(* PLC project PLC411_AI, home PLC411_AI 1 *)
(* stored: creationDateTime 2023-04-11T09:59:45, productRelease 0, modificationDateTime 2023-04-11T09:59:45, version 1 *)

(* Установка режима работы аналогового входа *)
FUNCTION_BLOCK AIMode
  VAR_INPUT
    AIn : BYTE := 0;  (* номер входа *)
    M : BYTE := 0;  (* режим работы *)
  END_VAR
  VAR_OUTPUT
    Om : BYTE := 0;  (* режим работы (установленный) *)
    Os : BYTE := 0;  (* код состояния входа *)
    Ok : BYTE := 0;  (* код результата исполнения блока *)
  END_VAR

            {extern void App_AIMode(AIMODE*);App_AIMode(data__);}

          
END_FUNCTION_BLOCK

(* Получение значения аналогового входа *)
FUNCTION_BLOCK AINorm
  VAR_INPUT
    AIn : BYTE := 0;  (* номер входа *)
  END_VAR
  VAR_OUTPUT
    Ov : REAL := 0.0;  (* значение *)
    Os : BYTE := 0;  (* код состояния *)
    Ok : BYTE := 0;  (* код результата исполнения блока *)
  END_VAR

            {extern void App_AINorm(AINORM*);App_AINorm(data__);}

          
END_FUNCTION_BLOCK
